FUNCTION_BLOCK Linearachse
VAR_INPUT
END_VAR
VAR_OUTPUT
END_VAR
VAR
END_VAR

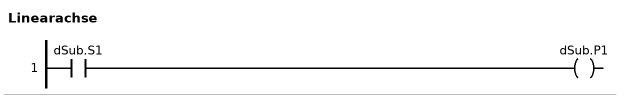
// NETWORK 1
dSub.P1 := dSub.S1;

END_FUNCTION_BLOCK

(* stored: Version 1.1.0.1, ProductVersion 3.1.4022.6
   POU Linearachse: Id {e7b84d25-bc80-459a-b78d-9976730e95b4}, SpecialFunc None *)
